(* Logix 5000 project; controller SX_V040001_C001 vendor 1 type 14 code 77 rev 16.23; software revision 16.04 *)
// SX_V04.00.01_C001

TASK InterruptTask (periodic, rate 5 ms, priority 10, watchdog 500 ms) : InterruptProgram
TASK MainTask (continuous, watchdog 500 ms) : MainProgram
TASK Task_100MS (periodic, rate 100 ms, priority 10, watchdog 500 ms) : Tastk_100MS

MODULES
   Controller : vendor 1 type 14 code 77 (CompactLogixL32EController 0, rev 16.23)
      LocalENB : 1769-L32E Ethernet Port (CompactLogixL32Ethernet 1, Ethernet 192.168.53.200, rev 16.1)
      Local : CompactBus (CompactVirtualAdapter 3, rev 16.1, Input RPI 2 ms)
         DI_2 : 1769-IQ32 (Compact 2, rev 3.1, Input RPI 2 ms)
         DI_1 : 1769-IQ32 (Compact 1, rev 3.1, Input RPI 2 ms)
         DI_3 : 1769-IQ32 (Compact 3, rev 3.1, Input RPI 2 ms)
         IF8_1 : 1769-MODULE (Compact 7, rev 1.1, Input RPI 2 ms)
         OF8C_1 : 1769-MODULE (Compact 8, rev 1.1, Output RPI 2 ms)
         DO_3 : vendor 1 type 7 code 73 (Compact 6, rev 3.1, Output RPI 2 ms)
         DO_2 : vendor 1 type 7 code 73 (Compact 5, rev 3.1, Output RPI 2 ms)
         DO_1 : vendor 1 type 7 code 73 (Compact 4, rev 3.1, Output RPI 2 ms)
END_MODULES

TYPE STRING_14 :
STRUCT
   LEN : DINT;
   DATA : SINT[14];
END_STRUCT
END_TYPE

VAR_GLOBAL   (* controller tags *)
   ALARM_BITS : INT[10] := ([4] := -32768);
   ALARM_BUFFER : INT[10] := ([0] := 4, [1] := 10, [2] := 11);
   ALL_KINDS : INT[90] := ([1] := 1, [2] := 3, [3] := 258, [4] := 530, [8] := 50, [9] := 99, [10] := 750, [11] := 600, [25] := 7270, [26] := 39, [27] := 7366, [28] := 40, [60] := 22660, [71] := 6);
   ANA_OUTPUT_SIM : INT[8] := ([1] := 2);
   average_current : DINT := 1045;
   Basic : INT;
   C_MINUTES : COUNTER := (PRE := 600, ACC := 274);
   C_SECONDS : COUNTER := (PRE := 10, ACC := 6);
   choco_control : PID := (CTL := 8426112, PE := 1, INI := 1, OLH := 1, DVPA := 1, PVHA := 1, SP := 9216.0, KP := 7.03, KI := 25.633333, MAXS := 27648.0, SO := 59.333332, MAXO := 59.333332, MINO := 10.0, UPD := 20.0, PV := 7366.0, ERR := 1850.0, OUT := 59.333332, MAXI := 27648.0, MAXCV := 27648.0, MAXTIE := 4095.0, DATA[0] := 50.400234, DATA[1] := -426.27313, DATA[2] := 7366.0, DATA[3] := 1850.0, DATA[4] := 9216.0, DATA[5] := 0.003616898, DATA[6] := 1.0, DATA[7] := 320.0, DATA[8] := 7.03, DATA[9] := 25.633333, DATA[11] := 7.03, DATA[12] := 0.0045708716, DATA[15] := 276.48, DATA[16] := 0.024420025);
   CMD : INT[36];
   command_number : INT := 55;
   command_type : DINT := 16#0000_c300;
   command_value : INT := 1;
   DATAOP : INT[10];
   DB_A_IO : INT[16] := ([0] := 26, [1] := 27, [4] := -25, [5] := -25, [7] := 2, [9] := 100);
   DB_D_IO : DINT[6] := ([0] := 571290609, [1] := 285250560, [2] := 992, [3] := 33882112, [4] := 939524096, [5] := 4456448);
   DB_D_IO_REVERSE : DINT[6] := ([0] := 220393779, [1] := 1114260, [2] := 57347, [3] := 84017152, [4] := 3670016, [5] := 1140850688);
   DIGI_OUTPUT_SIM : DINT[3] := ([0] := 33882112, [1] := 134217728);
   DIGI_OUTPUT_SIM_REVERSE : DINT[3] := ([0] := 84017152, [1] := 524288);
   DRIVE : INT[32] := ([7] := 11059, [8] := 13824, [9] := 27648, [10] := 210, [14] := 2000, [15] := 245, [17] := 14);
   Drive_diff_rpm_real : REAL;
   DRIVE_INTERVAL : INT[8];
   Drive_set_prop_rpm_real : REAL;
   EMPTYING : INT[18] := ([1] := 24, [3] := 45, [5] := 569, [8] := 49, [9] := 27648, [11] := 27648, [15] := 823, [16] := 34, [17] := 33);
   FP_ALARM_EXIST : BOOL := 1;
   FP_ALARM_RESET : BOOL;
   G_AInput : DINT[8] := ([0] := 7271, [1] := 7366, [2] := -26, [3] := -60, [4] := -6912, [5] := -6912, [6] := -10, [7] := 570);
   G_AOutput : DINT[8] := ([1] := 27648);
   G_DInput : DINT[3] := ([0] := 571290609, [1] := 285250560, [2] := 992);
   G_DOutput : DINT[3] := ([0] := 33882112, [1] := 939524096, [2] := 4456448);
   HANDSHAKE_VISIWIN : INT[3];
   loading : INT[19] := ([1] := 5888);
   louvre : INT[11] := ([3] := 641, [4] := 10);
   m_alarm_exist : BOOL := 1;
   m_alarm_horn : BOOL := 1;
   m_battery_low : BOOL;
   m_element_fault_reset : BOOL;
   m_notstop : BOOL;
   m_on_off_line : BOOL;
   m_power_up : BOOL;
   M_SIMU_ON_OFF : BOOL;
   M_VKE_1 : BOOL := 1;
   MESSAGE_BITS : INT[8] := ([0] := 3088);
   METERING : INT[44] := ([3] := 992, [40] := 511);
   METERING_PULSE : DINT[14];
   Min_Counter : DINT := 23;
   mw_major_fault : DINT;
   mw_minor_fault : DINT := 16;
   mw_temp : DINT := 47;
   negi_param398 : DINT;
   negi_param61 : DINT := -10;
   NOTDOS : INT[6];
   PARAM_VISIWIN_PART_1 : INT[101] := ([1] := 1, [2] := 5, [3] := 470, [4] := 60, [22] := 45, [24] := 45, [26] := 45, [27] := 10, [28] := 10, [29] := 10, [34] := 1, [60] := 1500, [61] := 10, [62] := 750, [63] := 30, [64] := 350, [65] := 350, [68] := 10, [100] := 1);
   PARAM_VISIWIN_PART_2 : INT[100] := ([4] := 10, [5] := 1, [7] := 5, [9] := 60, [10] := 10, [12] := 30, [13] := 10, [17] := 1, [18] := 5, [22] := 10, [24] := 5, [25] := 1, [27] := 5, [28] := 1, [30] := 5, [31] := 1, [33] := 5, [34] := 1, [36] := 5, [37] := 1, [39] := 6, [40] := 5, [41] := 20, [43] := 1000, [44] := 6, [45] := 5, [46] := 20, [48] := 1000, [50] := 5, [51] := 20, [53] := 1000, [55] := 5, [56] := 20, [58] := 1000, [60] := 5, [61] := 20, [63] := 1000, [65] := 5, [66] := 20, [67] := 1, [69] := 1000, [71] := 5, [73] := 5, [74] := 20, [75] := 1, [77] := 1000, [79] := 5, [81] := 5, [82] := 20, [83] := 1, [85] := 1000, [87] := 5, [89] := 5, [90] := 20, [91] := 1, [93] := 1000, [95] := 5, [99] := 6);
   PARAM_VISIWIN_PART_3 : INT[100] := ([0] := 1, [2] := 1000, [3] := 10, [6] := 5, [9] := 5, [10] := 20, [19] := 6, [20] := 1, [22] := 1000, [23] := 10, [26] := 5, [29] := 5, [30] := 20, [39] := 6, [40] := 1, [42] := 1000, [43] := 10, [46] := 5, [49] := 5, [50] := 20, [59] := 6, [60] := 1, [62] := 1000, [63] := 10, [66] := 5, [69] := 5, [70] := 20, [79] := 6, [80] := 1, [82] := 1000, [83] := 10, [86] := 5, [89] := 5, [90] := 20);
   PARAM_VISIWIN_PART_4 : INT[100] := ([2] := 99, [3] := 30, [4] := 99, [5] := 5, [6] := 120, [7] := 120, [8] := 5, [11] := 1, [12] := 1, [13] := 5, [39] := 1800, [40] := 33, [42] := 2, [43] := 703, [44] := 1538, [46] := 20, [47] := 89, [48] := 15, [81] := 30, [85] := 2000, [87] := 120, [88] := 300, [90] := 10, [91] := 60, [92] := 1, [93] := 1, [94] := 5, [95] := 5, [96] := 5, [98] := 7);
   PARAM_VISIWIN_PART_5 : INT[100] := ([0] := 60, [1] := 1, [2] := 45, [4] := 1, [5] := 120, [6] := 99, [12] := 4, [13] := 20, [16] := 15, [17] := 20, [18] := 30, [24] := 50, [25] := 5, [29] := 200, [33] := 5, [35] := 5, [41] := 100, [42] := 150, [43] := 5, [44] := 100, [45] := 100);
   PARAMETER : INT[501] := ([0] := 31, [1] := 1, [2] := 5, [3] := 470, [4] := 60, [22] := 45, [24] := 45, [26] := 45, [27] := 10, [28] := 10, [29] := 10, [34] := 1, [60] := 1500, [61] := 10, [62] := 750, [63] := 30, [64] := 350, [65] := 350, [68] := 10, [100] := 1, [105] := 10, [106] := 1, [108] := 5, [110] := 60, [111] := 10, [113] := 30, [114] := 10, [118] := 1, [119] := 5, [123] := 10, [125] := 5, [126] := 1, [128] := 5, [129] := 1, [131] := 5, [132] := 1, [134] := 5, [135] := 1, [137] := 5, [138] := 1, [140] := 6, [141] := 5, [142] := 20, [144] := 1000, [145] := 6, [146] := 5, [147] := 20, [149] := 1000, [151] := 5, [152] := 20, [154] := 1000, [156] := 5, [157] := 20, [159] := 1000, [161] := 5, [162] := 20, [164] := 1000, [166] := 5, [167] := 20, [168] := 1,
        [170] := 1000, [172] := 5, [174] := 5, [175] := 20, [176] := 1, [178] := 1000, [180] := 5, [182] := 5, [183] := 20, [184] := 1, [186] := 1000, [188] := 5, [190] := 5, [191] := 20, [192] := 1, [194] := 1000, [196] := 5, [200] := 6, [201] := 1, [203] := 1000, [204] := 10, [207] := 5, [210] := 5, [211] := 20, [220] := 6, [221] := 1, [223] := 1000, [224] := 10, [227] := 5, [230] := 5, [231] := 20, [240] := 6, [241] := 1, [243] := 1000, [244] := 10, [247] := 5, [250] := 5, [251] := 20, [260] := 6, [261] := 1, [263] := 1000, [264] := 10, [267] := 5, [270] := 5, [271] := 20, [280] := 6, [281] := 1, [283] := 1000, [284] := 10, [287] := 5, [290] := 5, [291] := 20, [303] := 99, [304] := 30, [305] := 99, [306] := 5, [307] := 120, [308] := 120, [309] := 5, [312] := 1,
        [313] := 1, [314] := 5, [340] := 1800, [341] := 33, [343] := 2, [344] := 703, [345] := 1538, [347] := 20, [348] := 89, [349] := 15, [382] := 30, [386] := 2000, [388] := 120, [389] := 300, [391] := 10, [392] := 60, [393] := 1, [394] := 1, [395] := 5, [396] := 5, [397] := 5, [399] := 7, [401] := 60, [402] := 1, [403] := 45, [405] := 1, [406] := 120, [407] := 99, [413] := 4, [414] := 20, [417] := 15, [418] := 20, [419] := 30, [425] := 50, [426] := 5, [430] := 200, [434] := 5, [436] := 5, [442] := 100, [443] := 150, [444] := 5, [445] := 100, [446] := 100);
   pointer_alarm_buffer : DINT := 3;
   pointer_bcc_in : DINT := 7;
   pointer_bcc_out : DINT := 7;
   pointer_bit_nr : DINT;
   pointer_dump_current : DINT;
   pointer_param_1 : DINT := 43;
   pointer_recipe : DINT := 57;
   pointer_recipe_line : DINT := 78;
   pointer_recipe_restart : DINT;
   pointer_recipe_test : DINT := 111;
   pointer_word_nr : DINT := 6;
   PULSE_ALARM_EXIST : BOOL;
   REC_NR_BCD_REMOTE : INT[5] := ([1] := 1);
   REC_NR_BCD_STRING : SINT[2];
   RECIPE_GENERAL : INT[405];
   RECIPE_VISIWIN_PART_1 : INT[100] := ([0] := 12336, [1] := 12336, [2] := 12336, [3] := 14640, [4] := 8275, [5] := 30030, [6] := 29555, [7] := 13088, [8] := 26416, [9] := 17184, [10] := 12589, [11] := 50, [12] := 12338, [13] := 12334, [14] := 11825, [15] := 13361, [16] := 13872, [17] := 12334, [18] := 11827, [19] := 12338, [20] := 25709, [21] := 6000, [22] := 80, [25] := 28, [27] := 15, [29] := 54, [30] := 42, [32] := 24, [35] := 10, [36] := 250, [38] := 35, [42] := 90, [44] := 52, [47] := 55, [48] := 45, [51] := 30, [54] := 2, [56] := 32, [59] := 55, [60] := 65, [63] := 30, [65] := 20, [66] := 2400, [68] := 10, [69] := 450, [72] := 300, [74] := 15, [75] := 210, [76] := 245, [78] := 15, [80] := 55, [81] := 45, [83] := 35, [87] := 5, [89] := 7, [90] := 2400, [93] := 30, [95] := 8, [96] := 1000, [98] := 59,
        [99] := 51);
   RECIPE_VISIWIN_PART_2 : INT[100] := ([1] := 54, [2] := 42, [4] := 53, [7] := 46);
   RECIPE_VISIWIN_PART_3 : INT[100];
   RECIPE_VISIWIN_PART_4 : INT[100];
   RECIPE_VISIWIN_PART_5 : INT[5];
   REMOTE_DATA_IN : INT[510] := ([0] := 512, [4] := -11520, [5] := -24320); {produced}
   REMOTE_DATA_OUT : INT[510] := ([0] := 20585, [2] := 1, [3] := 41, [4] := -22190, [5] := -24320, [6] := -8191, [7] := 1285, [8] := 1877, [9] := 1, [10] := 14, [11] := 4168, [14] := 525, [15] := 2057, [16] := 2, [18] := 79, [19] := 22660, [54] := 99, [55] := 50, [56] := 39, [58] := 40, [59] := 89, [60] := 100, [62] := 750, [63] := 600, [74] := 45, [87] := 6, [88] := 6, [89] := 6, [90] := 6, [91] := 6, [92] := 79, [97] := 2564, [98] := 11, [126] := 823); {produced}
   REMOTE_RECIPE : INT[405];
   REMOTE_SYSTEM : INT[38] := ([0] := 41, [1] := -24320, [2] := 7, [4] := 20585, [6] := 512);
   RM_CMD : INT[9] := ([1] := 16159, [2] := 496, [3] := 1920);
   s_bcc : INT := -22190;
   SOFTRELEASE_NUMBER : STRING_14 := 'V04.00.01_C001';
   STATUS_GENERAL : INT[135] := ([0] := -8191, [1] := 1285, [2] := 1877, [3] := 1, [4] := 14, [5] := 4168, [8] := 525, [9] := 2057, [10] := 2, [12] := 79, [13] := 22660, [48] := 99, [49] := 50, [50] := 39, [52] := 40, [53] := 89, [54] := 100, [56] := 750, [57] := 600, [68] := 45, [81] := 6, [82] := 6, [83] := 6, [84] := 6, [85] := 6, [86] := 79, [91] := 2564, [92] := 11, [120] := 823);
   STATUS_SEND_PART_1 : INT[135] := ([0] := -8191, [1] := 1285, [2] := 1877, [3] := 1, [4] := 14, [5] := 4168, [8] := 525, [9] := 2057, [10] := 2, [12] := 79, [13] := 22660, [48] := 99, [49] := 50, [50] := 39, [52] := 40, [53] := 89, [54] := 100, [56] := 750, [57] := 600, [68] := 45, [81] := 6, [82] := 6, [83] := 6, [84] := 6, [85] := 6, [86] := 79, [91] := 2564, [92] := 11, [120] := 823);
   T_ACT_DATA_RESET : TIMER := (PRE := 5000);
   T_AIR_EXH_FAN : TIMER := (PRE := 5000);
   T_AIR_IN_FAN : TIMER := (PRE := 5000);
   T_AIR_IN_HEATING : TIMER := (PRE := 5000);
   T_AIR_PRESSURE : TIMER := (PRE := 30000);
   T_BEARING_LUBR : TIMER := (PRE := 20000);
   T_CHOCO_PRESS_LOW : TIMER;
   T_CHOCO_PRESSURE : TIMER;
   T_CHOCO_PUMP : TIMER := (PRE := 5000);
   T_CONTR_CLFA_ACLFA : TIMER := (PRE := 10000);
   T_CONTR_CURR_SPEED : TIMER;
   T_COOLING_VALVE : TIMER;
   T_COVER_DOM : TIMER;
   T_CURRENT_AUTO : TIMER;
   T_CURRENT_CL : TIMER;
   T_CURRENT_EM_METER : TIMER;
   T_DEL_DATA : TIMER := (PRE := 10000);
   T_DELAY_BROKEN_AI_0 : TIMER := (PRE := 5000);
   T_DELAY_BROKEN_AI_1 : TIMER := (PRE := 5000);
   T_DELAY_BROKEN_AI_2 : TIMER := (PRE := 5000);
   T_DELAY_BROKEN_AI_3 : TIMER := (PRE := 5000);
   T_DELAY_BROKEN_AI_4 : TIMER := (PRE := 5000);
   T_DELAY_BROKEN_AI_5 : TIMER := (PRE := 5000);
   T_DELAY_BROKEN_AI_6 : TIMER := (PRE := 5000);
   T_DELAY_BROKEN_AI_7 : TIMER := (PRE := 5000);
   T_DELAY_COOLING_FAN : TIMER := (PRE := 600000);
   T_DELAY_SLOW_FAST : TIMER := (PRE := 1000);
   T_DELAY_SOFTSTART : TIMER := (PRE := 2000);
   T_DELTA_EM_METER : TIMER := (PRE := 300000);
   T_DRIVE_START_WARN : TIMER := (PRE := 5000);
   T_ELEKTR_HEAT : TIMER := (PRE := 5000);
   T_HEATING_VALVE : TIMER := (PRE := 2000, ACC := 1614, EN := 1, TT := 1);
   T_INLETT_VALVE : TIMER := (PRE := 30000);
   T_INTERN_CIRCLE : TIMER := (PRE := 99000);
   T_INTERVAL_HOUD_CL : TIMER := (PRE := 900000);
   T_LIVEBIT_OFF : TIMER := (PRE := 2000);
   T_LIVEBIT_ON : TIMER := (PRE := 2000, ACC := 253, EN := 1, TT := 1);
   T_LOADING_RELEASE : TIMER := (PRE := 5000, ACC := 5000, EN := 1, DN := 1);
   T_LOUVRE : TIMER := (PRE := 20000);
   T_MAX_CURRENT : TIMER := (PRE := 60000);
   T_MET10_END : TIMER := (PRE := 10000);
   T_MET11_END : TIMER := (PRE := 10000);
   T_MET12_END : TIMER := (PRE := 10000);
   T_MET13_END : TIMER := (PRE := 10000);
   T_MET14_END : TIMER := (PRE := 10000);
   T_MET1_END : TIMER := (PRE := 10000);
   T_MET2_END : TIMER := (PRE := 10000);
   T_MET3_END : TIMER := (PRE := 10000);
   T_MET4_END : TIMER := (PRE := 10000);
   T_MET5_END : TIMER := (PRE := 10000);
   T_MET6_END : TIMER := (PRE := 10000);
   T_MET7_END : TIMER := (PRE := 10000);
   T_MET8_END : TIMER := (PRE := 10000);
   T_MET9_END : TIMER := (PRE := 10000);
   T_MET_VALVE_1 : TIMER;
   T_MET_VALVE_10 : TIMER;
   T_MET_VALVE_11 : TIMER;
   T_MET_VALVE_12 : TIMER;
   T_MET_VALVE_13 : TIMER;
   T_MET_VALVE_14 : TIMER;
   T_MET_VALVE_2 : TIMER;
   T_MET_VALVE_3 : TIMER;
   T_MET_VALVE_4 : TIMER;
   T_MET_VALVE_5 : TIMER;
   T_MET_VALVE_6 : TIMER;
   T_MET_VALVE_7 : TIMER;
   T_MET_VALVE_8 : TIMER;
   T_MET_VALVE_9 : TIMER;
   T_MIN_ACTION_TIME : TIMER := (PRE := 5000);
   T_OUTLET_CLOSE : TIMER := (PRE := 99000, ACC := 99005);
   T_OUTLETT_VALVE : TIMER := (PRE := 60000);
   T_PULSE_HOUD_CL : TIMER := (PRE := 20000);
   T_RPM_EM_METER : TIMER;
   T_RUN_OUT_CHOCOPUMP : TIMER := (PRE := 300000);
   T_SAMPLER_OPEN : TIMER := (PRE := 120000);
   T_SCRAPER : TIMER := (PRE := 5000);
   T_START_ALARM : TIMER := (PRE := 200000);
   T_STUFFINGBOX_LUBR : TIMER := (PRE := 20000);
   T_TEMP_EM_METER : TIMER;
   T_WATER_NIVEAU : TIMER := (PRE := 99000);
   T_WATERPUMP : TIMER := (PRE := 5000);
   TEMP : INT[14] := ([1] := 4096, [4] := 5, [5] := 40, [6] := 89, [8] := 100, [9] := 65, [11] := 17, [13] := 2000);
   temp_bcc_in : DINT := 54016;
   temp_bcc_out : DINT := 43346;
   TEMP_REAL : REAL[22] := ([0] := 16404.48, [1] := 9216.0, [2] := 16404.48, [3] := 7271.0, [4] := 7366.0, [5] := 18.0, [6] := 0.55, [8] := 2000.0, [9] := 7.03, [10] := 25.633333, [12] := 20000.0, [13] := 10.0, [14] := 59.333332, [16] := 27648.002, [17] := 65.0, [18] := 17.0);
   TIMER_CHOCO_CONTR : TIMER := (PRE := 20000, ACC := 18049, EN := 1, TT := 1);
   TIMER_WATER_CONTR : TIMER := (PRE := 2000, ACC := 1604, EN := 1, TT := 1);
   water_control : PID := (CTL := 8426112, PE := 1, INI := 1, OLH := 1, DVPA := 1, PVHA := 1, SP := 16404.48, KP := 18.0, KI := 0.55, MAXS := 27648.0, SO := 100.0, MAXO := 100.0, MINO := -100.0, UPD := 2.0, PV := 7270.0, ERR := 9134.48, OUT := 100.0, MAXI := 27648.0, MAXCV := 27648.0, MAXTIE := 4095.0, DATA[0] := 96.01676, DATA[1] := -420.7176, DATA[2] := 7270.0, DATA[3] := 9134.48, DATA[4] := 16404.48, DATA[5] := 0.003616898, DATA[6] := 1.0, DATA[7] := 32.0, DATA[8] := 18.0, DATA[9] := 0.55, DATA[11] := 18.0, DATA[12] := 0.54545456, DATA[15] := 276.48, DATA[16] := 0.024420025);
   Z15 : COUNTER := (PRE := 120);
   Z16 : COUNTER := (PRE := 120);
   Z17 : COUNTER := (PRE := 120, ACC := 449, DN := 1);
   Z18 : COUNTER := (PRE := 120);
   Z19 : COUNTER := (PRE := 10);
   Z20 : COUNTER;
   Z21 : COUNTER := (PRE := 20);
   Z22 : COUNTER;
   Z23 : COUNTER;
   Z24 : COUNTER;
   Z25 : COUNTER;
   Z26 : COUNTER := (PRE := 20);
   Z27 : COUNTER := (PRE := 20);
   Z28 : COUNTER := (PRE := 20);
   Z29 : COUNTER := (PRE := 20);
   Z30 : COUNTER;
   Z31 : COUNTER;
   Z32 : COUNTER := (PRE := 10);
   Z33 : COUNTER;
   Z34 : COUNTER := (PRE := 20);
   Z35 : COUNTER;
   Z36 : COUNTER;
   Z37 : COUNTER;
   Z38 : COUNTER;
   Z39 : COUNTER;
   Z40 : COUNTER;
   Z41 : COUNTER;
   Z42 : COUNTER;
   Z43 : COUNTER;
   Z44 : COUNTER;
   Z45 : COUNTER;
   Z46 : COUNTER;
   Z47 : COUNTER;
   Z48 : COUNTER;
   Z49 : COUNTER;
   Z50 : COUNTER;
   Z_LIVE_COUNT : COUNTER := (PRE := 6);
END_VAR

PROGRAM InterruptProgram   (* main routine InterruptRoutine *)

ROUTINE InterruptRoutine   (* ladder *)
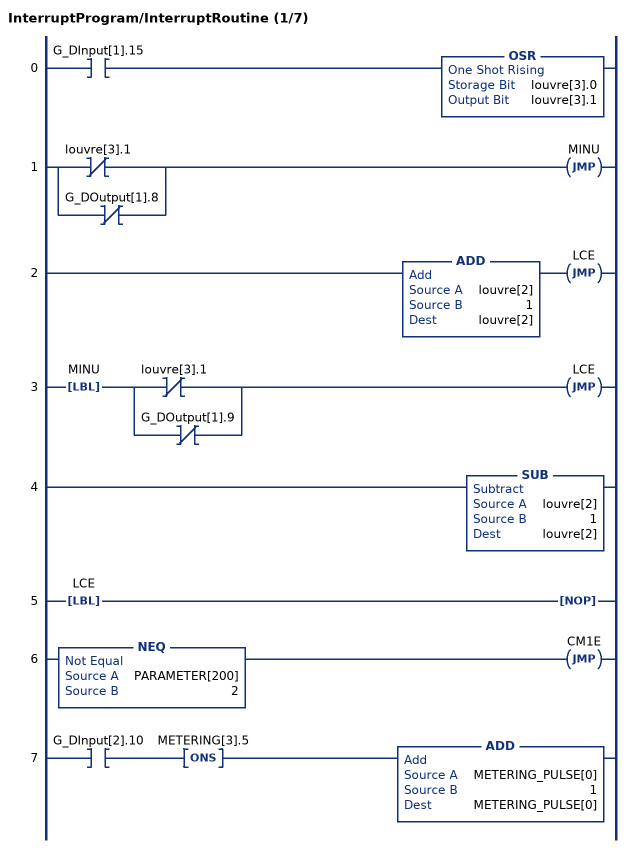
   0: XIC(G_DInput[1].15)OSR(louvre[3].0,louvre[3].1);
   1: [XIO(louvre[3].1) ,XIO(G_DOutput[1].8) ]JMP(MINU);
   2: ADD(louvre[2],1,louvre[2])JMP(LCE);
   3: LBL(MINU)[XIO(louvre[3].1) ,XIO(G_DOutput[1].9) ]JMP(LCE);
   4: SUB(louvre[2],1,louvre[2]);
   5: LBL(LCE)NOP();
   6: NEQ(PARAMETER[200],2)JMP(CM1E);
   7: XIC(G_DInput[2].10)ONS(METERING[3].5)ADD(METERING_PULSE[0],1,METERING_PULSE[0]);
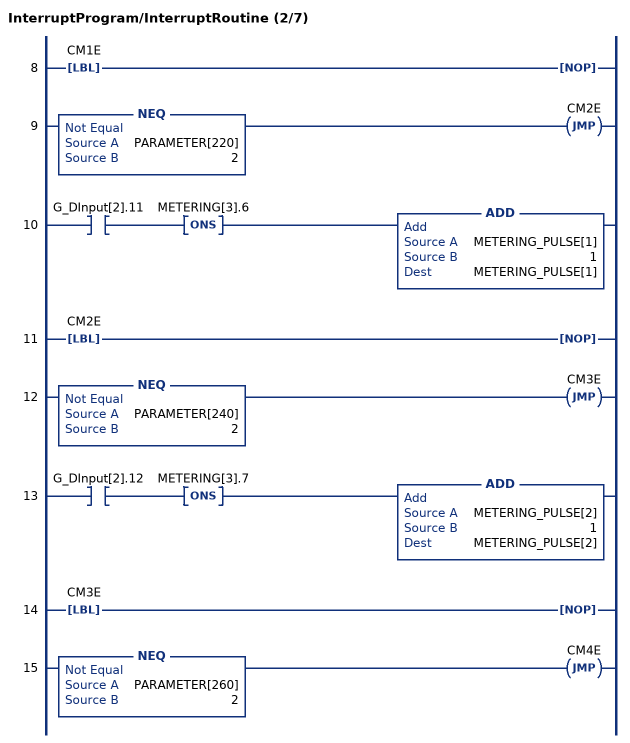
   8: LBL(CM1E)NOP();
   9: NEQ(PARAMETER[220],2)JMP(CM2E);
   10: XIC(G_DInput[2].11)ONS(METERING[3].6)ADD(METERING_PULSE[1],1,METERING_PULSE[1]);
   11: LBL(CM2E)NOP();
   12: NEQ(PARAMETER[240],2)JMP(CM3E);
   13: XIC(G_DInput[2].12)ONS(METERING[3].7)ADD(METERING_PULSE[2],1,METERING_PULSE[2]);
   14: LBL(CM3E)NOP();
   15: NEQ(PARAMETER[260],2)JMP(CM4E);
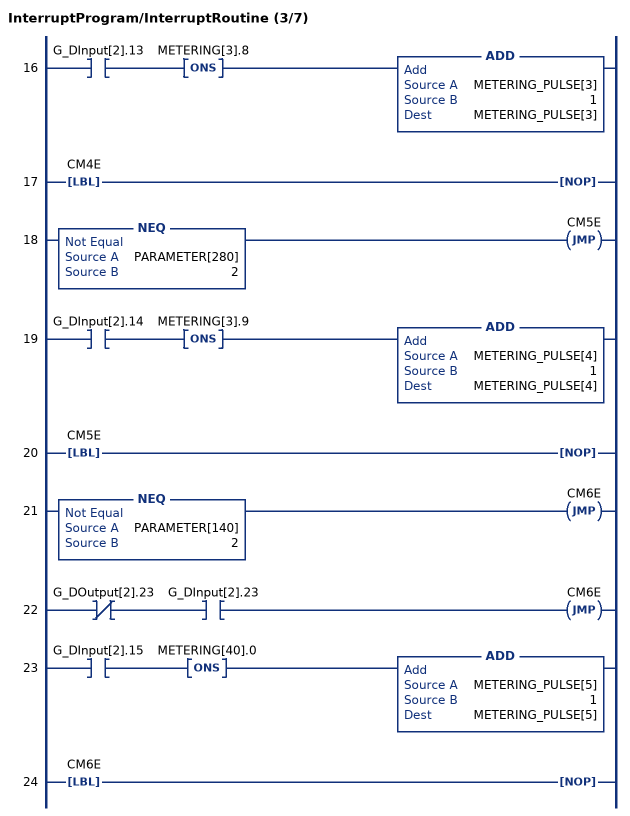
   16: XIC(G_DInput[2].13)ONS(METERING[3].8)ADD(METERING_PULSE[3],1,METERING_PULSE[3]);
   17: LBL(CM4E)NOP();
   18: NEQ(PARAMETER[280],2)JMP(CM5E);
   19: XIC(G_DInput[2].14)ONS(METERING[3].9)ADD(METERING_PULSE[4],1,METERING_PULSE[4]);
   20: LBL(CM5E)NOP();
   21: NEQ(PARAMETER[140],2)JMP(CM6E);
   22: XIO(G_DOutput[2].23)XIC(G_DInput[2].23)JMP(CM6E);
   23: XIC(G_DInput[2].15)ONS(METERING[40].0)ADD(METERING_PULSE[5],1,METERING_PULSE[5]);
   24: LBL(CM6E)NOP();
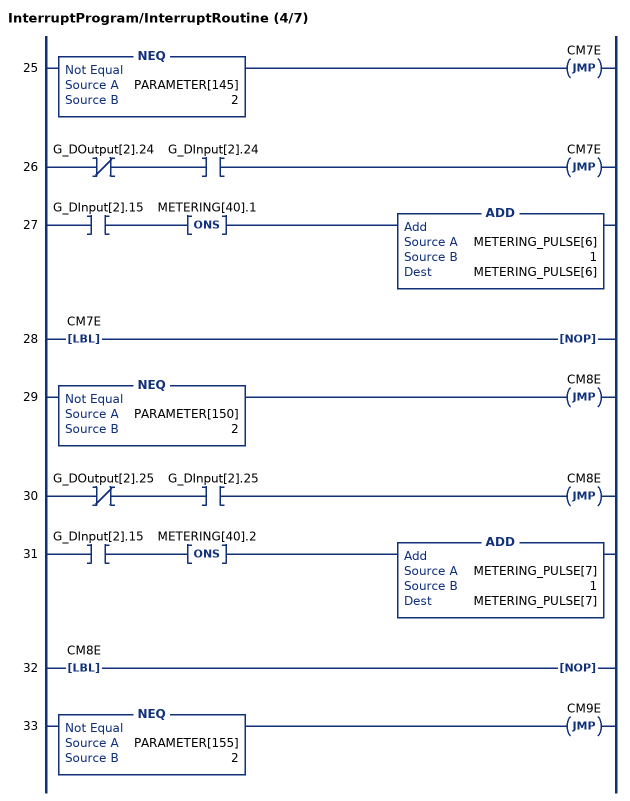
   25: NEQ(PARAMETER[145],2)JMP(CM7E);
   26: XIO(G_DOutput[2].24)XIC(G_DInput[2].24)JMP(CM7E);
   27: XIC(G_DInput[2].15)ONS(METERING[40].1)ADD(METERING_PULSE[6],1,METERING_PULSE[6]);
   28: LBL(CM7E)NOP();
   29: NEQ(PARAMETER[150],2)JMP(CM8E);
   30: XIO(G_DOutput[2].25)XIC(G_DInput[2].25)JMP(CM8E);
   31: XIC(G_DInput[2].15)ONS(METERING[40].2)ADD(METERING_PULSE[7],1,METERING_PULSE[7]);
   32: LBL(CM8E)NOP();
   33: NEQ(PARAMETER[155],2)JMP(CM9E);
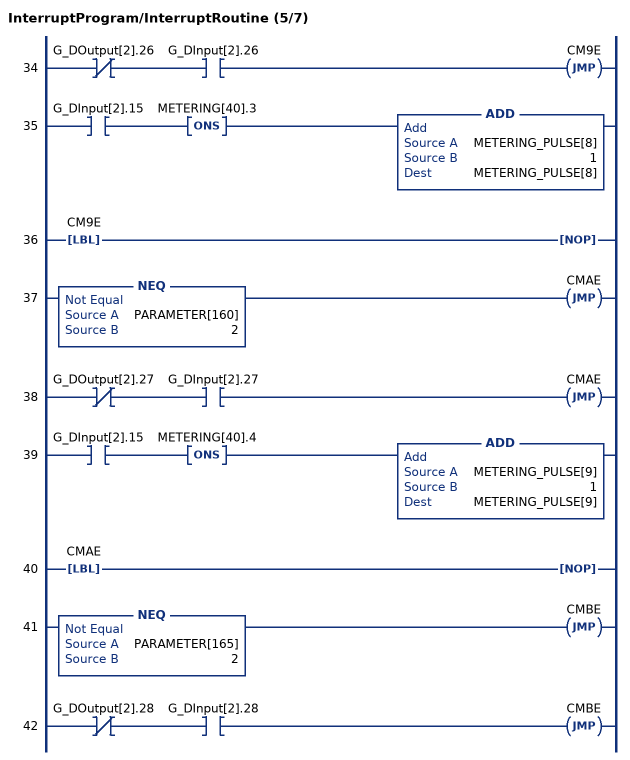
   34: XIO(G_DOutput[2].26)XIC(G_DInput[2].26)JMP(CM9E);
   35: XIC(G_DInput[2].15)ONS(METERING[40].3)ADD(METERING_PULSE[8],1,METERING_PULSE[8]);
   36: LBL(CM9E)NOP();
   37: NEQ(PARAMETER[160],2)JMP(CMAE);
   38: XIO(G_DOutput[2].27)XIC(G_DInput[2].27)JMP(CMAE);
   39: XIC(G_DInput[2].15)ONS(METERING[40].4)ADD(METERING_PULSE[9],1,METERING_PULSE[9]);
   40: LBL(CMAE)NOP();
   41: NEQ(PARAMETER[165],2)JMP(CMBE);
   42: XIO(G_DOutput[2].28)XIC(G_DInput[2].28)JMP(CMBE);
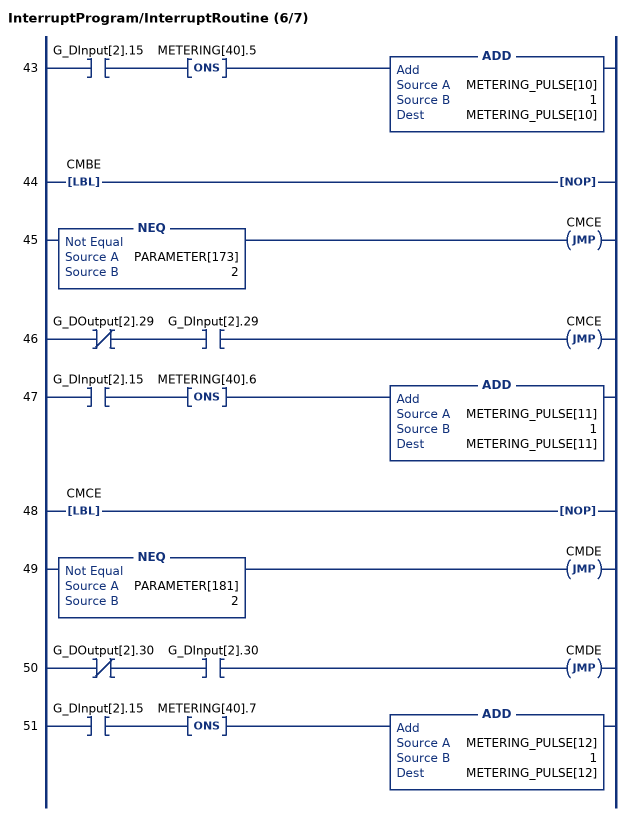
   43: XIC(G_DInput[2].15)ONS(METERING[40].5)ADD(METERING_PULSE[10],1,METERING_PULSE[10]);
   44: LBL(CMBE)NOP();
   45: NEQ(PARAMETER[173],2)JMP(CMCE);
   46: XIO(G_DOutput[2].29)XIC(G_DInput[2].29)JMP(CMCE);
   47: XIC(G_DInput[2].15)ONS(METERING[40].6)ADD(METERING_PULSE[11],1,METERING_PULSE[11]);
   48: LBL(CMCE)NOP();
   49: NEQ(PARAMETER[181],2)JMP(CMDE);
   50: XIO(G_DOutput[2].30)XIC(G_DInput[2].30)JMP(CMDE);
   51: XIC(G_DInput[2].15)ONS(METERING[40].7)ADD(METERING_PULSE[12],1,METERING_PULSE[12]);
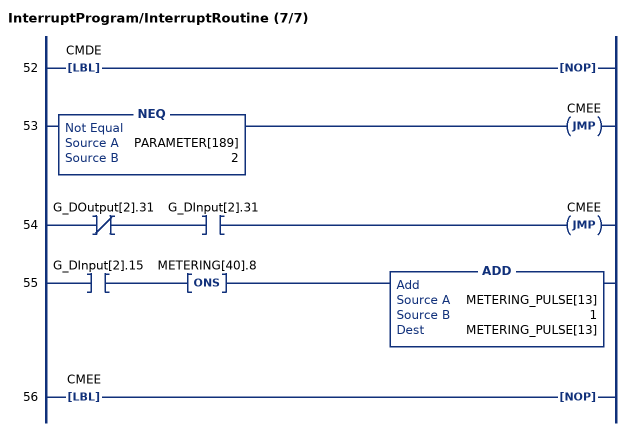
   52: LBL(CMDE)NOP();
   53: NEQ(PARAMETER[189],2)JMP(CMEE);
   54: XIO(G_DOutput[2].31)XIC(G_DInput[2].31)JMP(CMEE);
   55: XIC(G_DInput[2].15)ONS(METERING[40].8)ADD(METERING_PULSE[13],1,METERING_PULSE[13]);
   56: LBL(CMEE)NOP();
END_ROUTINE
END_PROGRAM

PROGRAM MainProgram   (* main routine MainRoutine *)
VAR
   testRick : BOOL := 1;
END_VAR

ROUTINE AirFan   (* ladder *)
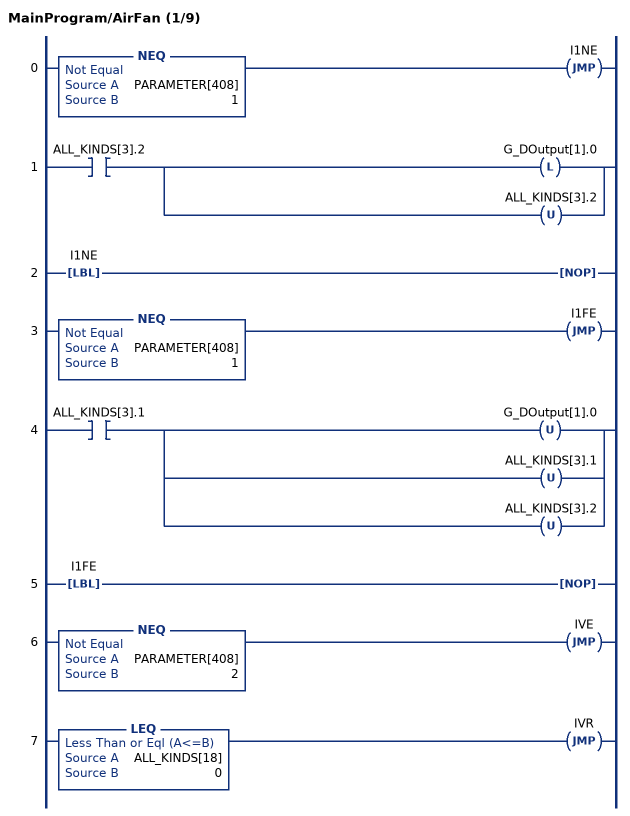
   0: NEQ(PARAMETER[408],1)JMP(I1NE);
   1: XIC(ALL_KINDS[3].2)[OTL(G_DOutput[1].0) ,OTU(ALL_KINDS[3].2) ];
   2: LBL(I1NE)NOP();
   3: NEQ(PARAMETER[408],1)JMP(I1FE);
   4: XIC(ALL_KINDS[3].1)[OTU(G_DOutput[1].0) ,OTU(ALL_KINDS[3].1) ,OTU(ALL_KINDS[3].2) ];
   5: LBL(I1FE)NOP();
   6: NEQ(PARAMETER[408],2)JMP(IVE);
   7: LEQ(ALL_KINDS[18],0)JMP(IVR);
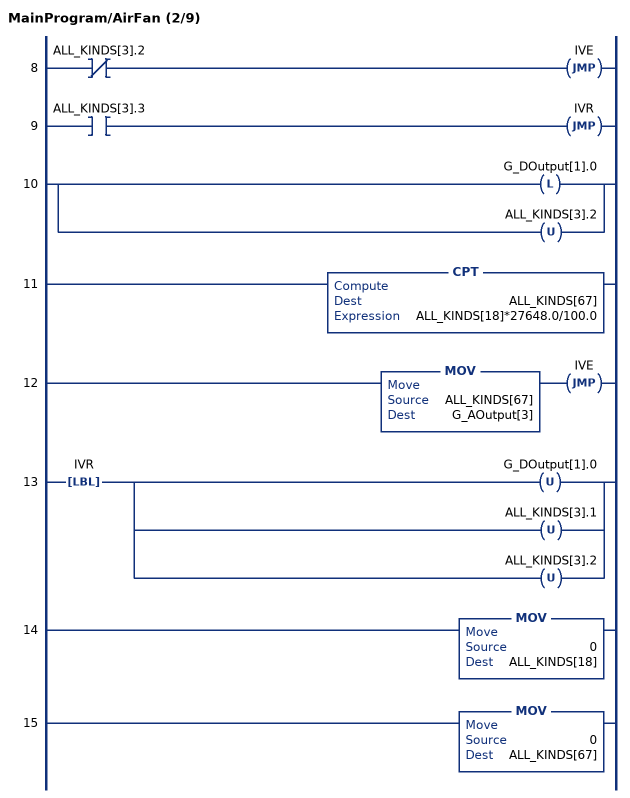
   8: XIO(ALL_KINDS[3].2)JMP(IVE);
   9: XIC(ALL_KINDS[3].3)JMP(IVR);
   10: [OTL(G_DOutput[1].0) ,OTU(ALL_KINDS[3].2) ];
   11: CPT(ALL_KINDS[67],ALL_KINDS[18]*27648.0/100.0);
   12: MOV(ALL_KINDS[67],G_AOutput[3])JMP(IVE);
   13: LBL(IVR)[OTU(G_DOutput[1].0) ,OTU(ALL_KINDS[3].1) ,OTU(ALL_KINDS[3].2) ];
   14: MOV(0,ALL_KINDS[18]);
   15: MOV(0,ALL_KINDS[67]);
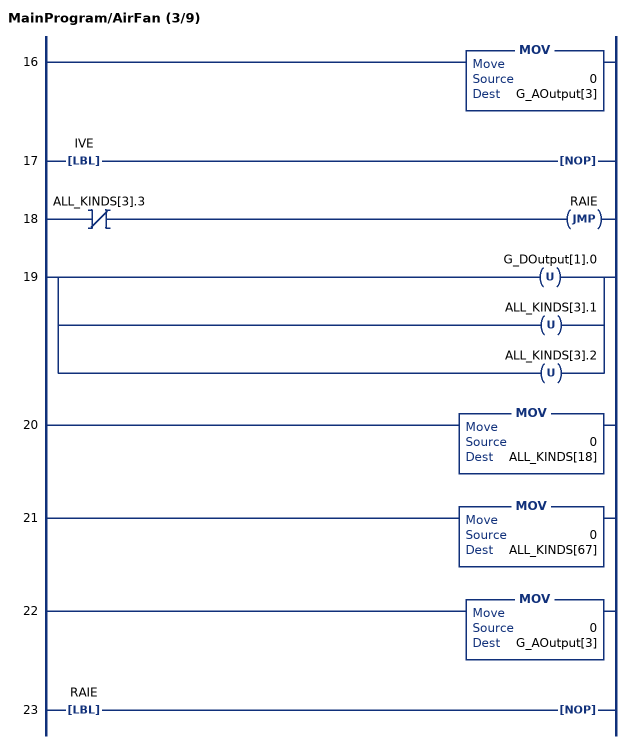
   16: MOV(0,G_AOutput[3]);
   17: LBL(IVE)NOP();
   18: XIO(ALL_KINDS[3].3)JMP(RAIE);
   19: [OTU(G_DOutput[1].0) ,OTU(ALL_KINDS[3].1) ,OTU(ALL_KINDS[3].2) ];
   20: MOV(0,ALL_KINDS[18]);
   21: MOV(0,ALL_KINDS[67]);
   22: MOV(0,G_AOutput[3]);
   23: LBL(RAIE)NOP();
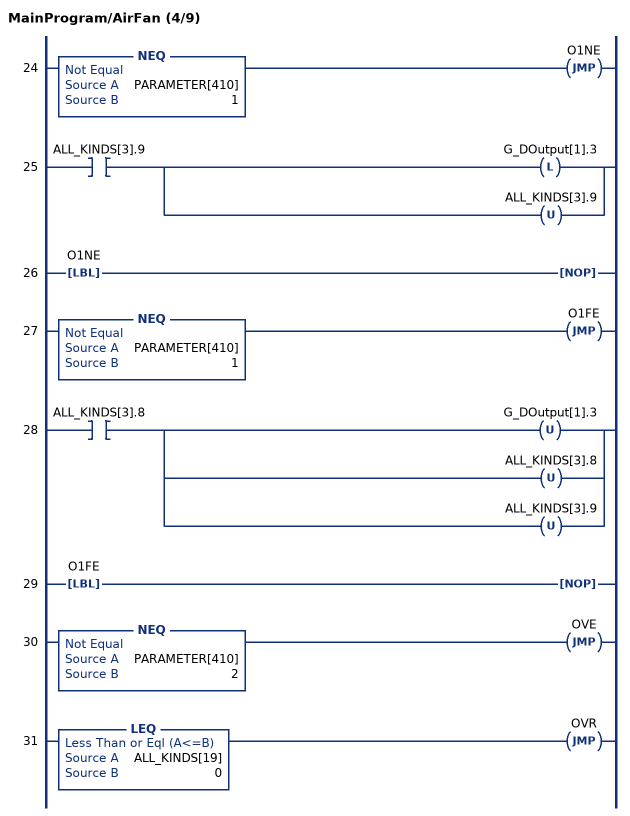
   24: NEQ(PARAMETER[410],1)JMP(O1NE);
   25: XIC(ALL_KINDS[3].9)[OTL(G_DOutput[1].3) ,OTU(ALL_KINDS[3].9) ];
   26: LBL(O1NE)NOP();
   27: NEQ(PARAMETER[410],1)JMP(O1FE);
   28: XIC(ALL_KINDS[3].8)[OTU(G_DOutput[1].3) ,OTU(ALL_KINDS[3].8) ,OTU(ALL_KINDS[3].9) ];
   29: LBL(O1FE)NOP();
   30: NEQ(PARAMETER[410],2)JMP(OVE);
   31: LEQ(ALL_KINDS[19],0)JMP(OVR);
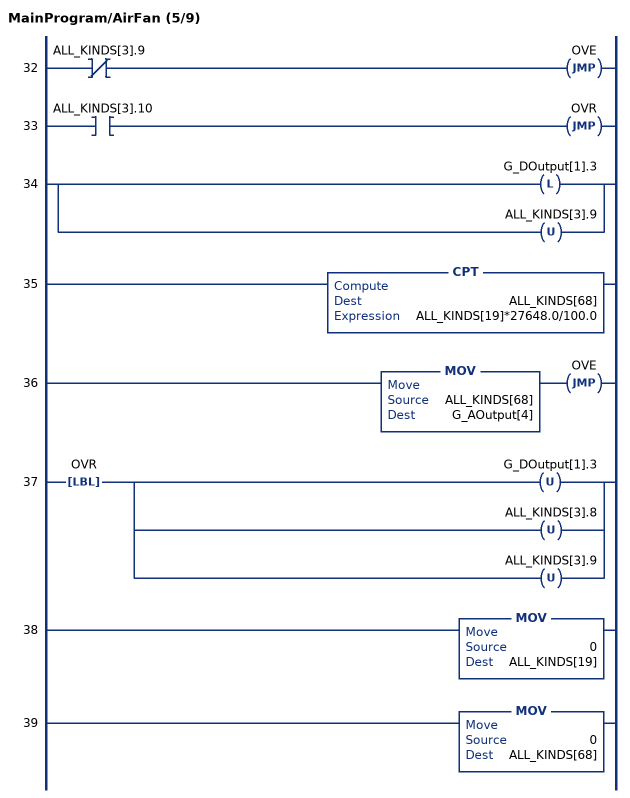
   32: XIO(ALL_KINDS[3].9)JMP(OVE);
   33: XIC(ALL_KINDS[3].10)JMP(OVR);
   34: [OTL(G_DOutput[1].3) ,OTU(ALL_KINDS[3].9) ];
   35: CPT(ALL_KINDS[68],ALL_KINDS[19]*27648.0/100.0);
   36: MOV(ALL_KINDS[68],G_AOutput[4])JMP(OVE);
   37: LBL(OVR)[OTU(G_DOutput[1].3) ,OTU(ALL_KINDS[3].8) ,OTU(ALL_KINDS[3].9) ];
   38: MOV(0,ALL_KINDS[19]);
   39: MOV(0,ALL_KINDS[68]);
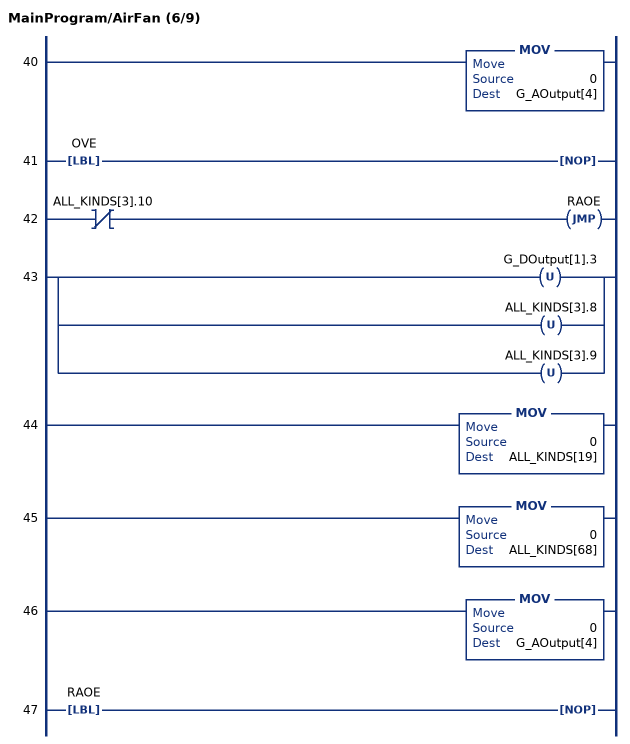
   40: MOV(0,G_AOutput[4]);
   41: LBL(OVE)NOP();
   42: XIO(ALL_KINDS[3].10)JMP(RAOE);
   43: [OTU(G_DOutput[1].3) ,OTU(ALL_KINDS[3].8) ,OTU(ALL_KINDS[3].9) ];
   44: MOV(0,ALL_KINDS[19]);
   45: MOV(0,ALL_KINDS[68]);
   46: MOV(0,G_AOutput[4]);
   47: LBL(RAOE)NOP();
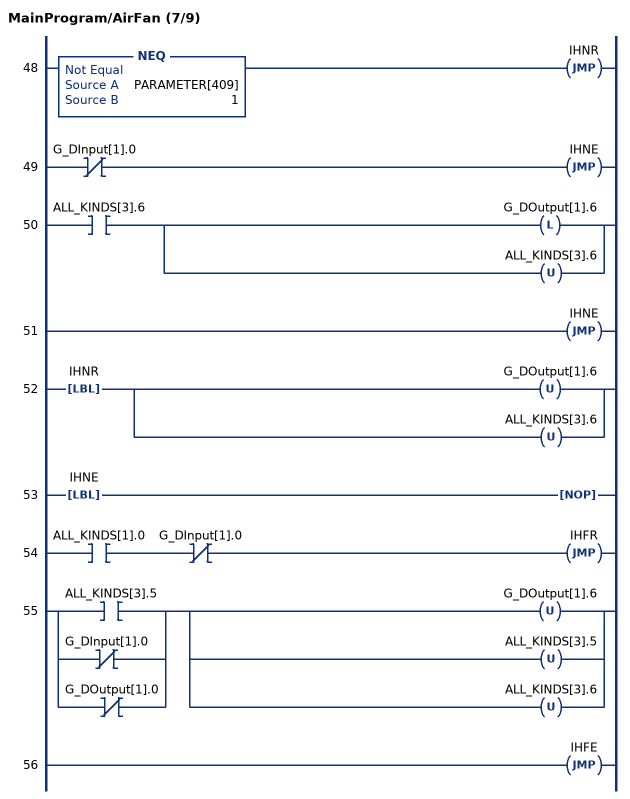
   48: NEQ(PARAMETER[409],1)JMP(IHNR);
   49: XIO(G_DInput[1].0)JMP(IHNE);
   50: XIC(ALL_KINDS[3].6)[OTL(G_DOutput[1].6) ,OTU(ALL_KINDS[3].6) ];
   51: JMP(IHNE);
   52: LBL(IHNR)[OTU(G_DOutput[1].6) ,OTU(ALL_KINDS[3].6) ];
   53: LBL(IHNE)NOP();
   54: XIC(ALL_KINDS[1].0)XIO(G_DInput[1].0)JMP(IHFR);
   55: [XIC(ALL_KINDS[3].5) ,XIO(G_DInput[1].0) ,XIO(G_DOutput[1].0) ][OTU(G_DOutput[1].6) ,OTU(ALL_KINDS[3].5) ,OTU(ALL_KINDS[3].6) ];
   56: JMP(IHFE);
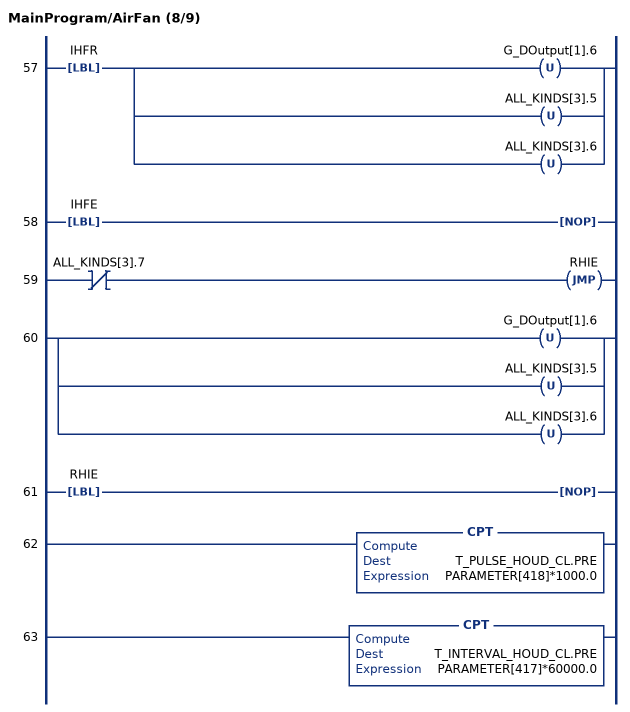
   57: LBL(IHFR)[OTU(G_DOutput[1].6) ,OTU(ALL_KINDS[3].5) ,OTU(ALL_KINDS[3].6) ];
   58: LBL(IHFE)NOP();
   59: XIO(ALL_KINDS[3].7)JMP(RHIE);
   60: [OTU(G_DOutput[1].6) ,OTU(ALL_KINDS[3].5) ,OTU(ALL_KINDS[3].6) ];
   61: LBL(RHIE)NOP();
   62: CPT(T_PULSE_HOUD_CL.PRE,PARAMETER[418]*1000.0);
   63: CPT(T_INTERVAL_HOUD_CL.PRE,PARAMETER[417]*60000.0);
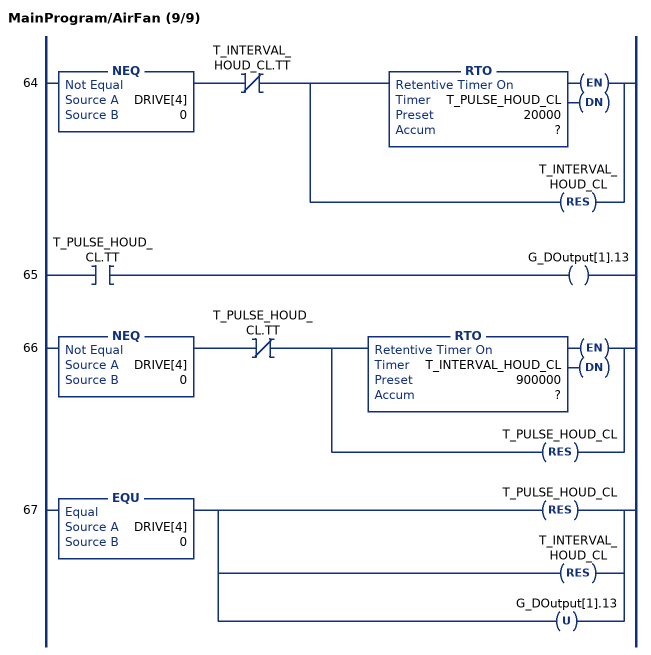
   64: NEQ(DRIVE[4],0)XIO(T_INTERVAL_HOUD_CL.TT)[RTO(T_PULSE_HOUD_CL,?,?) ,RES(T_INTERVAL_HOUD_CL) ];
   65: XIC(T_PULSE_HOUD_CL.TT)OTE(G_DOutput[1].13);
   66: NEQ(DRIVE[4],0)XIO(T_PULSE_HOUD_CL.TT)[RTO(T_INTERVAL_HOUD_CL,?,?) ,RES(T_PULSE_HOUD_CL) ];
   67: EQU(DRIVE[4],0)[RES(T_PULSE_HOUD_CL) ,RES(T_INTERVAL_HOUD_CL) ,OTU(G_DOutput[1].13) ];
END_ROUTINE

ROUTINE AlarmBitToNumber   (* ladder *)
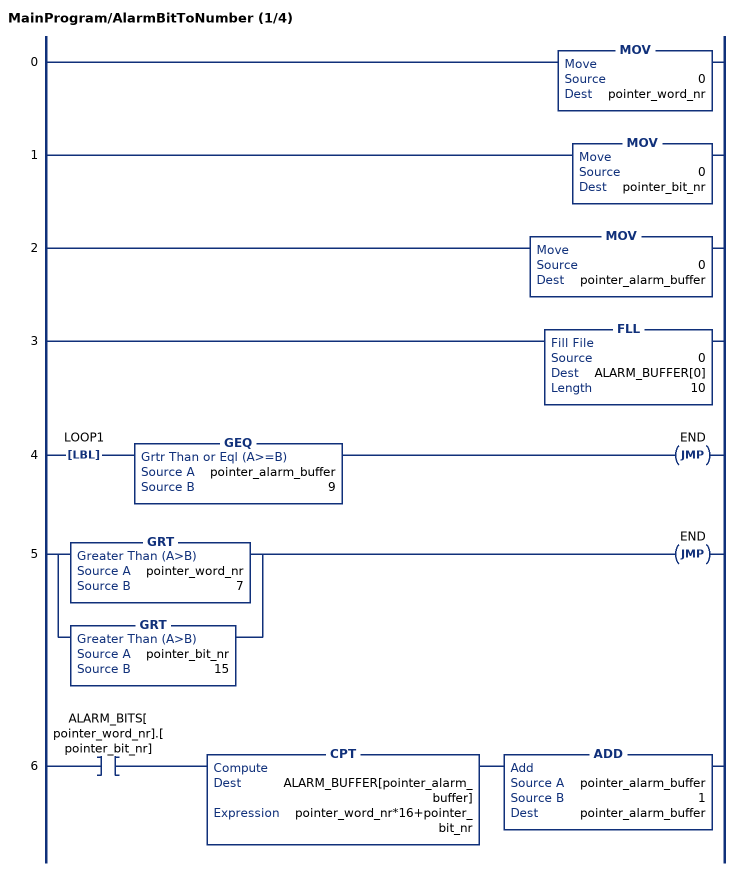
   0: MOV(0,pointer_word_nr);
   1: MOV(0,pointer_bit_nr);
   2: MOV(0,pointer_alarm_buffer);
   3: FLL(0,ALARM_BUFFER[0],10);
   4: LBL(LOOP1)GEQ(pointer_alarm_buffer,9)JMP(END);
   5: [GRT(pointer_word_nr,7) ,GRT(pointer_bit_nr,15) ]JMP(END);
   6: XIC(ALARM_BITS[pointer_word_nr].[pointer_bit_nr])CPT(ALARM_BUFFER[pointer_alarm_buffer],pointer_word_nr*16+pointer_bit_nr)ADD(pointer_alarm_buffer,1,pointer_alarm_buffer);
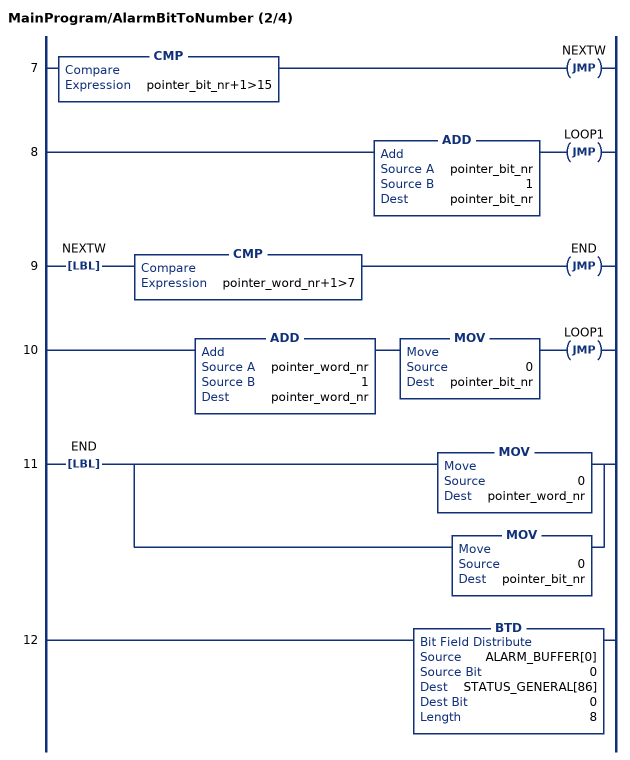
   7: CMP(pointer_bit_nr+1>15)JMP(NEXTW);
   8: ADD(pointer_bit_nr,1,pointer_bit_nr)JMP(LOOP1);
   9: LBL(NEXTW)CMP(pointer_word_nr+1>7)JMP(END);
   10: ADD(pointer_word_nr,1,pointer_word_nr)MOV(0,pointer_bit_nr)JMP(LOOP1);
   11: LBL(END)[MOV(0,pointer_word_nr) ,MOV(0,pointer_bit_nr) ];
   12: BTD(ALARM_BUFFER[0],0,STATUS_GENERAL[86],0,8);
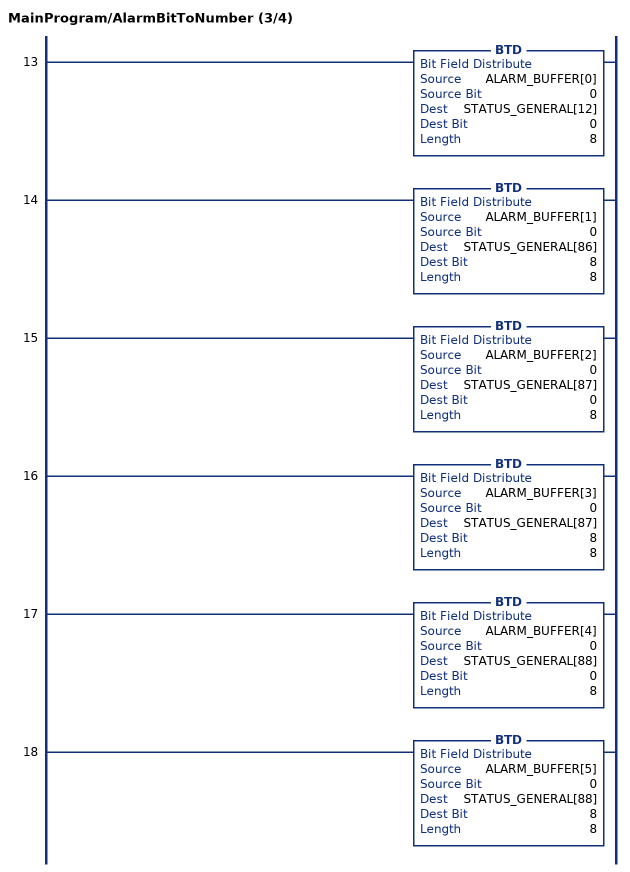
   13: BTD(ALARM_BUFFER[0],0,STATUS_GENERAL[12],0,8);
   14: BTD(ALARM_BUFFER[1],0,STATUS_GENERAL[86],8,8);
   15: BTD(ALARM_BUFFER[2],0,STATUS_GENERAL[87],0,8);
   16: BTD(ALARM_BUFFER[3],0,STATUS_GENERAL[87],8,8);
   17: BTD(ALARM_BUFFER[4],0,STATUS_GENERAL[88],0,8);
   18: BTD(ALARM_BUFFER[5],0,STATUS_GENERAL[88],8,8);
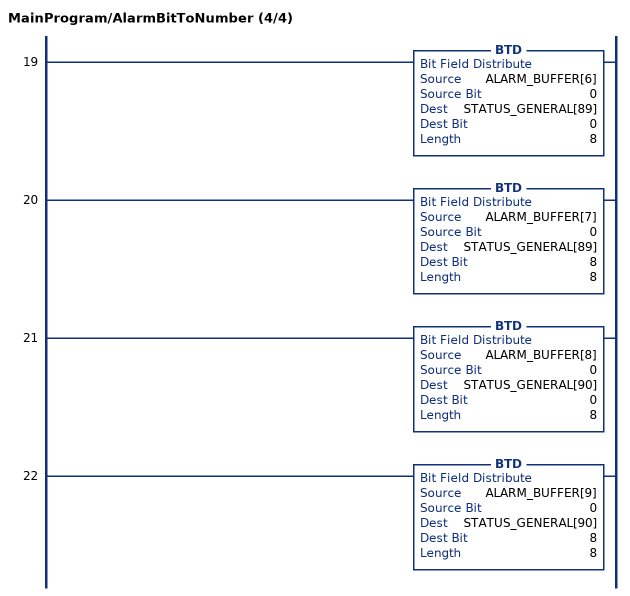
   19: BTD(ALARM_BUFFER[6],0,STATUS_GENERAL[89],0,8);
   20: BTD(ALARM_BUFFER[7],0,STATUS_GENERAL[89],8,8);
   21: BTD(ALARM_BUFFER[8],0,STATUS_GENERAL[90],0,8);
   22: BTD(ALARM_BUFFER[9],0,STATUS_GENERAL[90],8,8);
END_ROUTINE
